// TIA Portal project "PLC2_Client_Sever" (V16)

(* hardware
DEVICE "S71500/ET200MP station_1"  S7-1500 station
   slot 0: "Rail_0"  Rack  6ES7 590-1***0-0AA0
   slot 1: "PLC_Client"  CPU 1512C-1 PN  6ES7 512-1CK01-0AB0  V2.8
      slot 3: "CPU display_1"  6ES7591-1AA00-0AA0
      slot 32768: "PROFINET interface_1"  X1
         slot 32769: "Port_1"  X1 P1
         slot 32770: "Port_2"  X1 P2
      slot 34817: "Virtual CP interface port_1"  Virtual CP interface port  Virtual CP interface port
DEVICE "S71500/ET200MP station_2"  S7-1500 station
   slot 0: "Rail_0"  Rack  6ES7 590-1***0-0AA0
   slot 1: "PLC_Server"  CPU 1512C-1 PN  6ES7 512-1CK01-0AB0  V2.8
      slot 3: "CPU display_1"  6ES7591-1AA00-0AA0
      slot 32768: "PROFINET interface_1"  X1
         slot 32769: "Port_1"  X1 P1
         slot 32770: "Port_2"  X1 P2
      slot 34817: "Virtual CP interface port_1"  Virtual CP interface port  Virtual CP interface port
*)

// ===== PLC "PLC_Client"  CPU 1512C-1 PN =====

VAR_GLOBAL   // PLC tag table "Default tag table"
   "System_Byte" AT %MB1 : Byte;
   "FirstScan" AT %M1.0 : Bool;
   "DiagStatusUpdate" AT %M1.1 : Bool;
   "AlwaysTRUE" AT %M1.2 : Bool;
   "AlwaysFALSE" AT %M1.3 : Bool;
   "System_Byte(1)" AT %MB1 : Byte;
   "Clock_Byte" AT %MB100 : Byte;
   "Clock_10Hz" AT %M100.0 : Bool;
   "Clock_5Hz" AT %M100.1 : Bool;
   "Clock_2.5Hz" AT %M100.2 : Bool;
   "Clock_2Hz" AT %M100.3 : Bool;
   "Clock_1.25Hz" AT %M100.4 : Bool;
   "Clock_1Hz" AT %M100.5 : Bool;
   "Clock_0.625Hz" AT %M100.6 : Bool;
   "Clock_0.5Hz" AT %M100.7 : Bool;
   "Tag_1" AT %MD10 : DWord;
   "Tag_2" AT %MW10 : Word;
   "Tag_3" AT %MW12 : Word;
   "Tag_4" AT %MW14 : Word;
   "Tag_5" AT %MW16 : Word;
   "Tag_6" AT %MW18 : Word;
   "Tag_7" AT %MW20 : Word;
   "Tag_8" AT %MW22 : Word;
   "Tag_9" AT %MW24 : Word;
   "Tag_10" AT %MD14 : Real;
   "Tag_11" AT %MD18 : Real;
   "Tag_12" AT %MD22 : Real;
END_VAR

DATA_BLOCK "Connection"   // DB1
{ S7_Optimized_Access := 'TRUE' }
VERSION : 0.1
   VAR
      ClientConnect : TCON_IP_v4;
   END_VAR
BEGIN
   ClientConnect.InterfaceId := 64;
   ClientConnect.ID := 1;
   ClientConnect.ActiveEstablished := 1;
   ClientConnect.RemoteAddress.ADDR[1] := 192;
   ClientConnect.RemoteAddress.ADDR[2] := 168;
   ClientConnect.RemoteAddress.ADDR[3] := 1;
   ClientConnect.RemoteAddress.ADDR[4] := 202;
   ClientConnect.RemotePort := 502;
END_DATA_BLOCK

DATA_BLOCK "DB_Client"   // DB3
{ S7_Optimized_Access := 'TRUE' }
VERSION : 0.1
   VAR
      DATA : Array[0..7] of Word;
   END_VAR
BEGIN
   DATA[0] := 0;
END_DATA_BLOCK

DATA_BLOCK "DB_Data"   // DB4
{ S7_Optimized_Access := 'TRUE' }
VERSION : 0.1
   VAR
      "DT" : Array[0..3] of Real;
   END_VAR
BEGIN
END_DATA_BLOCK

ORGANIZATION_BLOCK "Main"   // OB1, LAD, ProgramCycle
TITLE = "Main Program Sweep (Cycle)"
{ S7_Optimized_Access := 'TRUE' }
VERSION : 0.1
   VAR_INPUT
      Initial_Call : Bool;   // Initial call of this OB
      Remanence : Bool;   // =True, if remanent data are available
   END_VAR
BEGIN

REGION Network 1
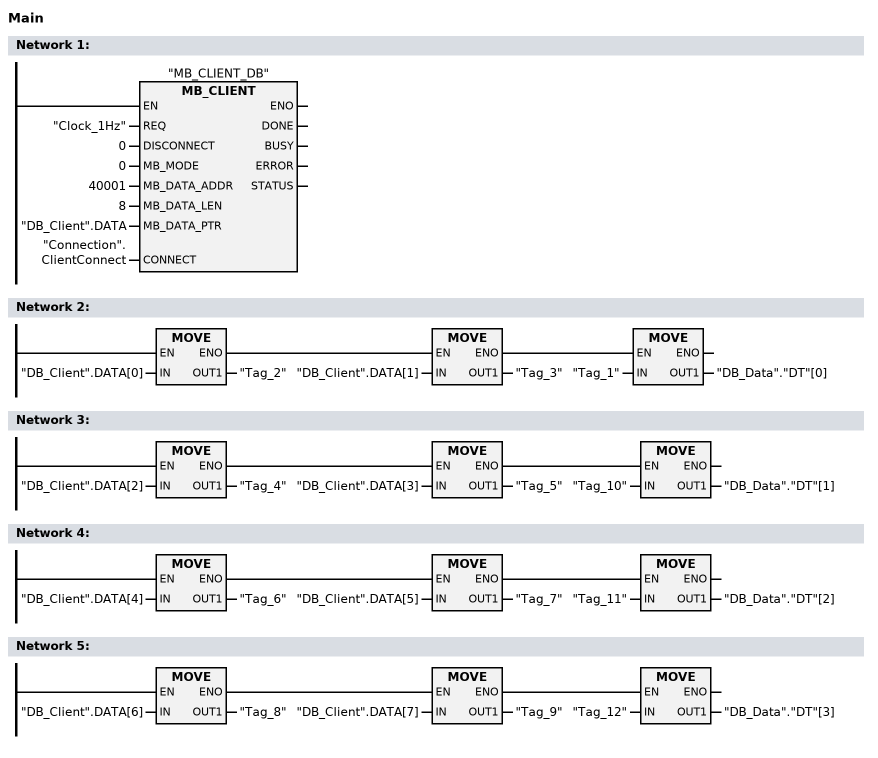
   "MB_CLIENT_DB"(REQ := "Clock_1Hz",   // MB_CLIENT
                  DISCONNECT := 0,
                  MB_MODE := 0,
                  MB_DATA_ADDR := 40001,
                  MB_DATA_LEN := 8,
                  MB_DATA_PTR := "DB_Client".DATA,
                  CONNECT := "Connection".ClientConnect);
END_REGION

REGION Network 2
   RUNG wire#powerrail
      Move(in := "DB_Client".DATA[0], out1 => "Tag_2")
      Move(in := "DB_Client".DATA[1], out1 => "Tag_3")
      Move(in := "Tag_1", out1 => "DB_Data"."DT"[0])
   END_RUNG
   // the same network as SCL:
   "Tag_2" := "DB_Client".DATA[0];
   "Tag_3" := "DB_Client".DATA[1];
   "DB_Data"."DT"[0] := "Tag_1";
END_REGION

REGION Network 3
   RUNG wire#powerrail
      Move(in := "DB_Client".DATA[2], out1 => "Tag_4")
      Move(in := "DB_Client".DATA[3], out1 => "Tag_5")
      Move(in := "Tag_10", out1 => "DB_Data"."DT"[1])
   END_RUNG
   // the same network as SCL:
   "Tag_4" := "DB_Client".DATA[2];
   "Tag_5" := "DB_Client".DATA[3];
   "DB_Data"."DT"[1] := "Tag_10";
END_REGION

REGION Network 4
   RUNG wire#powerrail
      Move(in := "DB_Client".DATA[4], out1 => "Tag_6")
      Move(in := "DB_Client".DATA[5], out1 => "Tag_7")
      Move(in := "Tag_11", out1 => "DB_Data"."DT"[2])
   END_RUNG
   // the same network as SCL:
   "Tag_6" := "DB_Client".DATA[4];
   "Tag_7" := "DB_Client".DATA[5];
   "DB_Data"."DT"[2] := "Tag_11";
END_REGION

REGION Network 5
   RUNG wire#powerrail
      Move(in := "DB_Client".DATA[6], out1 => "Tag_8")
      Move(in := "DB_Client".DATA[7], out1 => "Tag_9")
      Move(in := "Tag_12", out1 => "DB_Data"."DT"[3])
   END_RUNG
   // the same network as SCL:
   "Tag_8" := "DB_Client".DATA[6];
   "Tag_9" := "DB_Client".DATA[7];
   "DB_Data"."DT"[3] := "Tag_12";
END_REGION
END_ORGANIZATION_BLOCK

// ===== PLC "PLC_Server"  CPU 1512C-1 PN =====

VAR_GLOBAL   // PLC tag table "Default tag table"
   "Tag_1" AT %MW10 : Word;
   "Tag_2" AT %MW12 : Word;
   "Tag_3" AT %MW14 : Word;
   "Tag_4" AT %MW22 : Word;
   "Tag_5" AT %MW18 : Word;
   "Clock_Byte" AT %MB100 : Byte;
   "Clock_10Hz" AT %M100.0 : Bool;
   "Clock_5Hz" AT %M100.1 : Bool;
   "Clock_2.5Hz" AT %M100.2 : Bool;
   "Clock_2Hz" AT %M100.3 : Bool;
   "Clock_1.25Hz" AT %M100.4 : Bool;
   "Clock_1Hz" AT %M100.5 : Bool;
   "Clock_0.625Hz" AT %M100.6 : Bool;
   "Clock_0.5Hz" AT %M100.7 : Bool;
   "Tag_6" AT %MD10 : DWord;
   "Tag_7" AT %M500.0 : Bool;
   "Tag_8" AT %MW16 : Word;
   "Tag_9" AT %MW24 : Word;
   "Tag_10" AT %MW20 : Word;
END_VAR

DATA_BLOCK "DB_Server"   // DB2
{ S7_Optimized_Access := 'TRUE' }
VERSION : 0.1
   VAR
      Data : Array[0..7] of Word;
   END_VAR
BEGIN
END_DATA_BLOCK

DATA_BLOCK "Server_connect"   // DB3
{ S7_Optimized_Access := 'TRUE' }
VERSION : 0.1
   VAR
      SV_connect : TCON_IP_v4;
   END_VAR
BEGIN
   SV_connect.InterfaceId := 64;
   SV_connect.ID := 1;
   SV_connect.ActiveEstablished := 0;
   SV_connect.LocalPort := 502;
END_DATA_BLOCK

ORGANIZATION_BLOCK "Main"   // OB1, LAD, ProgramCycle
TITLE = "Main Program Sweep (Cycle)"
{ S7_Optimized_Access := 'TRUE' }
VERSION : 0.1
   VAR_INPUT
      Initial_Call : Bool;   // Initial call of this OB
      Remanence : Bool;   // =True, if remanent data are available
   END_VAR
   VAR_TEMP   // added for the SCL form of the ladder/FBD networks
      _w1 : Bool;
   END_VAR
BEGIN

REGION Network 1
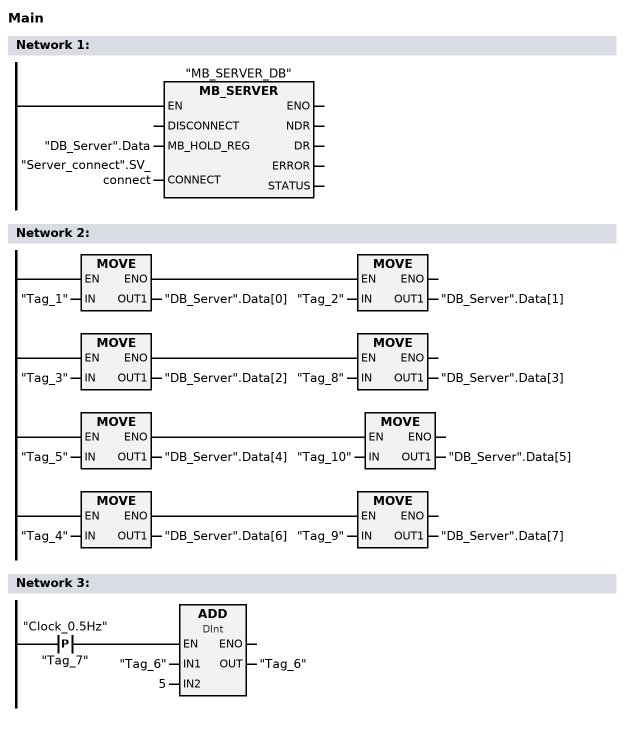
   "MB_SERVER_DB"(MB_HOLD_REG := "DB_Server".Data, CONNECT := "Server_connect".SV_connect);   // MB_SERVER
END_REGION

REGION Network 2
   RUNG wire#powerrail
      Move(in := "Tag_1", out1 => "DB_Server".Data[0])
      Move(in := "Tag_2", out1 => "DB_Server".Data[1])
   END_RUNG
   RUNG wire#powerrail
      Move(in := "Tag_3", out1 => "DB_Server".Data[2])
      Move(in := "Tag_8", out1 => "DB_Server".Data[3])
   END_RUNG
   RUNG wire#powerrail
      Move(in := "Tag_5", out1 => "DB_Server".Data[4])
      Move(in := "Tag_10", out1 => "DB_Server".Data[5])
   END_RUNG
   RUNG wire#powerrail
      Move(in := "Tag_4", out1 => "DB_Server".Data[6])
      Move(in := "Tag_9", out1 => "DB_Server".Data[7])
   END_RUNG
   // the same network as SCL:
   "DB_Server".Data[0] := "Tag_1";
   "DB_Server".Data[1] := "Tag_2";
   "DB_Server".Data[2] := "Tag_3";
   "DB_Server".Data[3] := "Tag_8";
   "DB_Server".Data[4] := "Tag_5";
   "DB_Server".Data[5] := "Tag_10";
   "DB_Server".Data[6] := "Tag_4";
   "DB_Server".Data[7] := "Tag_9";
END_REGION

REGION Network 3
   RUNG wire#powerrail
      P_Contact(operand := "Clock_0.5Hz", bit := "Tag_7")
      { S7_Templates := "SrcType := DInt" } Add(in1 := "Tag_6", in2 := 5, out => "Tag_6")
   END_RUNG
   // the same network as SCL:
   #_w1 := "Clock_0.5Hz" AND NOT "Tag_7";   // rising edge of "Clock_0.5Hz"
   "Tag_7" := "Clock_0.5Hz";
   IF #_w1 THEN "Tag_6" := "Tag_6" + 5; END_IF;
END_REGION
END_ORGANIZATION_BLOCK